Universal Robots PolyScope program: cottonbot.urp

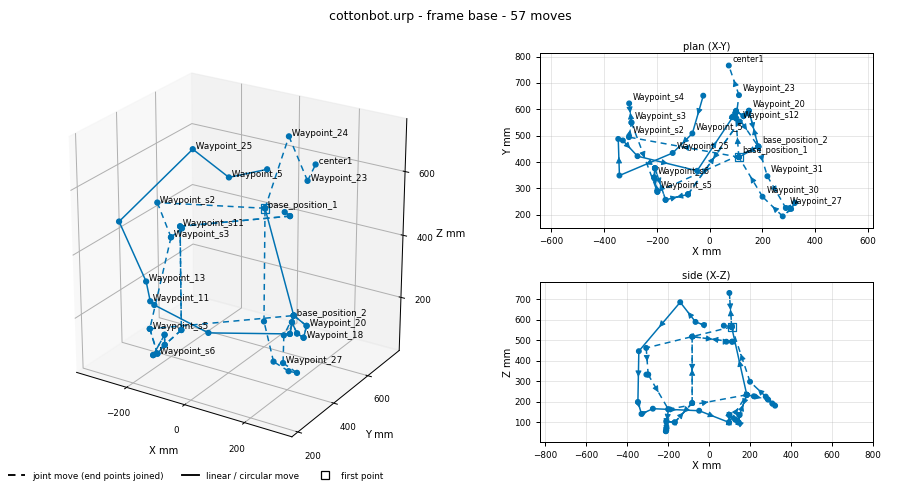
[picture p0: tool path of cottonbot.urp in frame base, 57 of 63 moves have a stored position in this frame; points joined in program order, loops and branches not executed]
Program cottonbot (installation=default directory=/programs/Nicolas_Arteaga/new folder createdIn=5.8.2.10297 lastSavedIn=5.12.4.1101661 robotSerialNumber=20225502378)
Calibrated DH parameters: a=[0.00022, -0.425328, -0.389701, 0.000059, 0.000065, 0]; d=[0.162608, 0.803456, 9.992211, -10.662202, 0.099702, 0.099559]; alpha=[1.570756, 0.001543, 0.004316, 1.570651, -1.570122, 0]; deltaTheta=[0, 0.002917, 0.116094, -0.119008, 0, -0.000001]
Robot Program (runOnlyOnce=true)
  'The whole program merged'
  Timer (action=Start) variable(name=timer_2)
  Timer (action=Start) variable(name=timer_3)
  'Now starts the Sugar Workflow'
  MoveJ speed 60 deg/s, acceleration 80 deg/s^2 (useActiveTCP=true) feature=Base
    Waypoint base_position_1: TCP in base x=110.873 y=418.875 z=565.206 mm, rx=-1.5602 ry=-0.9891 rz=-1.3624 rad; joints [200.91, -129.117, 99.415, 36.172, 41.428, 90] deg; TCP offset x=0 y=0 z=191.5 mm, rx=0 ry=0 rz=0 rad
    Waypoint Waypoint_s2: TCP in base x=-305.749 y=494.617 z=462.545 mm, rx=-1.1337 ry=-1.2693 rz=-1.1298 rad; joints [300.263, -100.211, 102.502, -1.736, 114.115, 89.999] deg; TCP offset x=0 y=0 z=191.5 mm, rx=0 ry=0 rz=0 rad
    URCap Gripper Activate (Robotiq_Grippers, Robotiq Inc.) dataModel(ResetAndActivateKey=false)
    URCap Gripper (Robotiq_Grippers, Robotiq Inc.) dataModel(position=20.0, force=0.0, speed=0.0, positionInDouble=20.0, forceInDouble=0.0, speedInDouble=0.0, slaveIds=[9], blocking=true)
    Waypoint Waypoint_s3: TCP in base x=-296.164 y=549.885 z=332.617 mm, rx=-1.2863 ry=-1.1731 rz=-1.2824 rad; joints [302.576, -85.481, 108.119, -21.976, 128.323, 90.062] deg
    Waypoint Waypoint_s4: TCP in base x=-304.886 y=622.528 z=332.693 mm, rx=-1.2845 ry=-1.1692 rz=-1.2825 rad; joints [298.729, -77.999, 99.501, -20.953, 124.442, 90.195] deg
    URCap Gripper (Robotiq_Grippers, Robotiq Inc.) dataModel(position=35.0, force=100.0, speed=100.0, positionInDouble=35.0, forceInDouble=100.0, speedInDouble=100.0, slaveIds=[9], blocking=true)
    Wait Sleep waitTime=0.5
    URCap Gripper (Robotiq_Grippers, Robotiq Inc.) dataModel(position=0.0, force=100.0, speed=0.0, positionInDouble=0.0, forceInDouble=100.0, speedInDouble=0.0, slaveIds=[9], blocking=true)
    Waypoint Waypoint_s3: TCP in base x=-296.164 y=549.885 z=332.617 mm, rx=-1.2863 ry=-1.1731 rz=-1.2824 rad; joints [302.576, -85.481, 108.119, -21.976, 128.323, 90.062] deg
    Waypoint Waypoint_s5: TCP in base x=-197.91 y=287.3 z=163.432 mm, rx=-1.5535 ry=0.1524 rz=-0.1096 rad; joints [326.967, -91.614, 148.2, -58.357, 156.715, 180] deg; TCP offset x=0 y=0 z=191.5 mm, rx=0 ry=0 rz=0 rad
    URCap Gripper (Robotiq_Grippers, Robotiq Inc.) dataModel(position=50.0, force=100.0, speed=0.0, positionInDouble=50.0, forceInDouble=100.0, speedInDouble=0.0, slaveIds=[9], blocking=true)
    Waypoint Waypoint_s6: TCP in base x=-209.858 y=341.762 z=56.515 mm, rx=-1.5807 ry=0.0548 rz=-0.0662 rad; joints [313.143, -65.937, 152.318, -85.713, 137.744, 180] deg; TCP offset x=0 y=0 z=191.5 mm, rx=0 ry=0 rz=0 rad
    Waypoint Waypoint_s7: TCP in base x=-207.363 y=377.054 z=70.962 mm, rx=-1.5764 ry=0.0343 rz=-0.0374 rad; joints [304.137, -69.797, 152.569, -82.518, 126.942, 179.974] deg; TCP offset x=0 y=0 z=191.5 mm, rx=0 ry=0 rz=0 rad
    URCap Gripper (Robotiq_Grippers, Robotiq Inc.) dataModel(position=100.0, force=100.0, speed=0.0, positionInDouble=100.0, forceInDouble=100.0, speedInDouble=0.0, slaveIds=[9], blocking=true)
    Waypoint Waypoint_s8: TCP in base x=-207.108 y=376.646 z=104.52 mm, rx=-1.5811 ry=0.0321 rz=-0.0396 rad; joints [304.156, -79.665, 151.838, -71.558, 126.955, 180.055] deg
    Waypoint Waypoint_s9: TCP in base x=-166.798 y=256.956 z=99.586 mm, rx=-1.5812 ry=0.0311 rz=-0.0496 rad; joints [323.963, -84.01, 161.527, -76.66, 147.1, 180] deg; TCP offset x=0 y=0 z=191.5 mm, rx=0 ry=0 rz=0 rad
    Waypoint Waypoint_s10: TCP in base x=-81.738 y=277.755 z=193.913 mm, rx=-1.6539 ry=-0.0026 rz=-1.0019 rad; joints [319.07, -96.736, 145.387, -56.678, 176.026, 135] deg; TCP offset x=0 y=0 z=191.5 mm, rx=0 ry=0 rz=0 rad
    Waypoint Waypoint_s11: TCP in base x=-81.724 y=277.748 z=517.554 mm, rx=-1.6566 ry=-0.0181 rz=-1.0161 rad; joints [319.137, -114.467, 104.986, 2.526, 175.909, 135] deg; TCP offset x=0 y=0 z=191.5 mm, rx=0 ry=0 rz=0 rad
    Waypoint Waypoint_s12: TCP in base x=113.097 y=553.265 z=492.993 mm, rx=-1.5561 ry=-0.4924 rz=-0.7353 rad; joints [227.113, -110.707, 105.414, 5.953, 56.661, 135.029] deg; TCP offset x=0 y=0 z=191.5 mm, rx=0 ry=0 rz=0 rad
    Waypoint Waypoint_s13: TCP in base x=85.146 y=570.31 z=492.98 mm, rx=-0.6297 ry=-2.0123 rz=-2.0637 rad; joints [234.679, -108.87, 104.254, 5.245, 64.223, 25.001] deg; TCP offset x=0 y=0 z=191.5 mm, rx=0 ry=0 rz=0 rad
    Waypoint Waypoint_s12: TCP in base x=113.097 y=553.265 z=492.993 mm, rx=-1.5561 ry=-0.4924 rz=-0.7353 rad; joints [227.113, -110.707, 105.414, 5.953, 56.661, 135.029] deg; TCP offset x=0 y=0 z=191.5 mm, rx=0 ry=0 rz=0 rad
    Waypoint Waypoint_s11: TCP in base x=-81.724 y=277.748 z=517.554 mm, rx=-1.6566 ry=-0.0181 rz=-1.0161 rad; joints [319.137, -114.467, 104.986, 2.526, 175.909, 135] deg; TCP offset x=0 y=0 z=191.5 mm, rx=0 ry=0 rz=0 rad
    Waypoint Waypoint_s10: TCP in base x=-81.738 y=277.755 z=193.913 mm, rx=-1.6539 ry=-0.0026 rz=-1.0019 rad; joints [319.07, -96.736, 145.387, -56.678, 176.026, 135] deg; TCP offset x=0 y=0 z=191.5 mm, rx=0 ry=0 rz=0 rad
    Waypoint Waypoint_s9: TCP in base x=-166.798 y=256.956 z=99.586 mm, rx=-1.5812 ry=0.0311 rz=-0.0496 rad; joints [323.963, -84.01, 161.527, -76.66, 147.1, 180] deg; TCP offset x=0 y=0 z=191.5 mm, rx=0 ry=0 rz=0 rad
    Waypoint Waypoint_s8: TCP in base x=-207.108 y=376.646 z=104.52 mm, rx=-1.5811 ry=0.0321 rz=-0.0396 rad; joints [304.156, -79.665, 151.838, -71.558, 126.955, 180.055] deg; TCP offset x=0 y=0 z=191.5 mm, rx=0 ry=0 rz=0 rad
    Waypoint Waypoint_s7: TCP in base x=-207.363 y=377.054 z=70.962 mm, rx=-1.5764 ry=0.0343 rz=-0.0374 rad; joints [304.137, -69.797, 152.569, -82.518, 126.942, 179.974] deg
    URCap Gripper (Robotiq_Grippers, Robotiq Inc.) dataModel(position=0.0, force=0.0, speed=100.0, positionInDouble=0.0, forceInDouble=0.0, speedInDouble=100.0, slaveIds=[9], blocking=true)
    Waypoint Waypoint_s6: TCP in base x=-209.858 y=341.762 z=56.515 mm, rx=-1.5807 ry=0.0548 rz=-0.0662 rad; joints [313.143, -65.937, 152.318, -85.713, 137.744, 180] deg; TCP offset x=0 y=0 z=191.5 mm, rx=0 ry=0 rz=0 rad
    Waypoint Waypoint_s5: TCP in base x=-197.91 y=287.3 z=163.432 mm, rx=-1.5535 ry=0.1524 rz=-0.1096 rad; joints [326.967, -91.614, 148.2, -58.357, 156.715, 180] deg; TCP offset x=0 y=0 z=191.5 mm, rx=0 ry=0 rz=0 rad
    Waypoint base_position_2: TCP in base x=184.715 y=458.614 z=234.006 mm, rx=-1.6866 ry=-0.757 rz=-1.7388 rad; joints [237.954, -104.402, 143.977, -41.546, 99.477, 90] deg; TCP offset x=0 y=0 z=191.5 mm, rx=0 ry=0 rz=0 rad
  'Now starts turning on the machine'
  MoveJ speed 60 deg/s, acceleration 80 deg/s^2 (useActiveTCP=true) feature=Base
    URCap Gripper (Robotiq_Grippers, Robotiq Inc.) dataModel(position=100.0, force=0.0, speed=100.0, positionInDouble=100.0, forceInDouble=0.0, speedInDouble=100.0, slaveIds=[9], blocking=true)
    Waypoint base_position_2: TCP in base x=184.715 y=458.614 z=234.006 mm, rx=-1.6866 ry=-0.757 rz=-1.7388 rad; joints [237.954, -104.402, 143.977, -41.546, 99.477, 90] deg
    Waypoint Waypoint_20: TCP in base x=148.965 y=594.736 z=135.542 mm, rx=-1.534 ry=-0.9908 rz=-1.4978 rad; joints [241.135, -76.483, 134.799, -57.047, 85.473, 90.096] deg; TCP offset x=0 y=0 z=191.5 mm, rx=0 ry=0 rz=0 rad
    Waypoint Waypoint_18: TCP in base x=144.729 y=585.254 z=99.641 mm, rx=-1.6452 ry=-1.0629 rz=-1.3952 rad; joints [240.345, -76.212, 134.041, -48.93, 84.034, 89.956] deg
    Waypoint Waypoint_6: TCP in base x=128.361 y=574.771 z=113.603 mm, rx=-1.6021 ry=-1.0547 rz=-1.4085 rad; joints [240.991, -78.96, 136.832, -51.045, 83.741, 89.995] deg
    Waypoint Waypoint_17: TCP in base x=99.779 y=593.316 z=135.031 mm, rx=-1.492 ry=-1.1083 rz=-1.3373 rad; joints [241.005, -80.644, 135.434, -49.386, 76.736, 90.11] deg
    Waypoint Waypoint_16: TCP in base x=97.63 y=585.581 z=99.564 mm, rx=-1.5888 ry=-1.15 rz=-1.2562 rad; joints [240.815, -78.841, 134.769, -44.332, 76.722, 90.097] deg
    Waypoint base_position_2: TCP in base x=184.715 y=458.614 z=234.006 mm, rx=-1.6866 ry=-0.757 rz=-1.7388 rad; joints [237.954, -104.402, 143.977, -41.546, 99.477, 90] deg; TCP offset x=0 y=0 z=191.5 mm, rx=0 ry=0 rz=0 rad
  'Now the stick Placement'
  MoveJ speed 60 deg/s, acceleration 80 deg/s^2 (useActiveTCP=true) feature=Base
    Waypoint base_position_2: TCP in base x=184.715 y=458.614 z=234.006 mm, rx=-1.6866 ry=-0.757 rz=-1.7388 rad; joints [237.954, -104.402, 143.977, -41.546, 99.477, 90] deg
    URCap Gripper Activate (Robotiq_Grippers, Robotiq Inc.) dataModel(ResetAndActivateKey=false)
    URCap Gripper (Robotiq_Grippers, Robotiq Inc.) dataModel(position=70.0, force=0.0, speed=100.0, positionInDouble=70.0, forceInDouble=0.0, speedInDouble=100.0, slaveIds=[9], blocking=true)
    Waypoint Waypoint_31: TCP in base x=219.073 y=346.37 z=226.939 mm, rx=-1.0793 ry=1.1503 rz=-0.4496 rad; joints [242.985, -108.839, 146.791, -38.8, 126.314, 210] deg; TCP offset x=0 y=0 z=191.5 mm, rx=0 ry=0 rz=0 rad
    Waypoint Waypoint_27: TCP in base x=288.911 y=225.994 z=210.348 mm, rx=-0.5682 ry=1.4712 rz=-0.493 rad; joints [230.777, -108.395, 149.908, -42.839, 137.738, 230] deg; TCP offset x=0 y=0 z=191.5 mm, rx=0 ry=0 rz=0 rad
    Waypoint stick1: TCP in base x=322.798 y=244.707 z=180.935 mm, rx=-0.6006 ry=1.5021 rz=-0.5325 rad; joints [227.883, -97.858, 147.006, -47.332, 135.838, 229.943] deg; TCP offset x=0 y=0 z=191.5 mm, rx=0 ry=0 rz=0 rad
    URCap Gripper (Robotiq_Grippers, Robotiq Inc.) dataModel(position=100.0, force=0.0, speed=0.0, positionInDouble=100.0, forceInDouble=0.0, speedInDouble=0.0, slaveIds=[9], blocking=true)
    Waypoint Waypoint_3: TCP in base x=308.934 y=222.719 z=191.895 mm, rx=-0.6005 ry=1.5021 rz=-0.5324 rad; joints [226.032, -105.235, 149.7, -42.849, 134.017, 229.721] deg
    Waypoint Waypoint_4: TCP in base x=277.219 y=194.361 z=225.221 mm, rx=-0.5767 ry=1.5048 rz=-0.5799 rad; joints [231.096, -114.882, 148.99, -33.185, 141.571, 228.474] deg
    Waypoint Waypoint_30: TCP in base x=200.562 y=268.796 z=297.612 mm, rx=-1.3009 ry=0.8471 rz=-0.8634 rad; joints [232.325, -138.788, 148.891, -15.287, 116.251, 180] deg; TCP offset x=0 y=0 z=191.5 mm, rx=0 ry=0 rz=0 rad
    Waypoint Waypoint_28: TCP in base x=110.872 y=418.885 z=565.169 mm, rx=-1.6121 ry=0.3611 rz=-0.2078 rad; joints [200.913, -129.115, 99.418, 36.172, 41.428, 180] deg; TCP offset x=0 y=0 z=191.5 mm, rx=0 ry=0 rz=0 rad
    Waypoint Waypoint_24: TCP in base x=99.712 y=565.5 z=730.734 mm, rx=-1.4619 ry=0.2517 rz=-0.2966 rad; joints [243.031, -99.822, 65.521, 28.761, 83.192, 180] deg; TCP offset x=0 y=0 z=191.5 mm, rx=0 ry=0 rz=0 rad
    Waypoint Waypoint_23: TCP in base x=111.331 y=653.695 z=566.749 mm, rx=-1.7943 ry=0.2693 rz=-0.1351 rad; joints [243.037, -87.632, 65.808, 35.91, 77.265, 180] deg; TCP offset x=0 y=0 z=191.5 mm, rx=0 ry=0 rz=0 rad
    Waypoint center1: TCP in base x=72.723 y=766.045 z=571.175 mm, rx=-1.5688 ry=-0.0203 rz=0.0146 rad; joints [244.553, -79.065, 65.7, 13.074, 63.165, 180.144] deg; TCP offset x=0 y=0 z=191.5 mm, rx=0 ry=0 rz=0 rad
  'Now Cotton Candy Creation'
  SuppressedNode
    radius := 0.149
  radius := 0.13
  height := 0.05
  SuppressedNode
    cold_start_wait := 101.25
  SuppressedNode
    start_wait := GP_int_in[0]
  SuppressedNode
    start_time := GP_int_in[1]
  SuppressedNode
    circle_time := GP_int_in[2]
  start_wait := 1
  start_time := 33.75
  circle_time := 3.75
  SuppressedNode
    cold_start_spin := 28
  SuppressedNode
    cold_start_spin := 100
  center := Joint_6_name
  bottom := pose_add(center, p[0, -radius, height, 0, 0, 0])
  right := pose_add(center, p[-radius, 0, -height, 0, 0, 0])
  top_circ := pose_add(center, p[0, radius, height, 0, 0, 0])
  left := pose_add(center, p[radius, 0, -height, 0, 0, 0])
  SuppressedNode
    diff := pose_sub(left,bottom )
  SuppressedNode
    Loop While (checkContinuously=false) expression=circles_no>0
      MoveP speed 250 mm/s, acceleration 1200 mm/s^2 (blendRadius=0.125 useActiveTCP=true) feature=Base
        Waypoint Waypoint (Variable): variable(name=bottom)
        CircleMove (OrientationMode=UNCONSTRAINED)
          Waypoint Waypoint (Variable): variable=left
          Waypoint Waypoint (Variable): variable(name=top_circ)
      MoveP speed 250 mm/s, acceleration 1200 mm/s^2 (blendRadius=0.025 useActiveTCP=true) feature=Base
        Waypoint Waypoint (Variable): variable=top_circ
        CircleMove (OrientationMode=UNCONSTRAINED)
          Waypoint Waypoint (Variable): variable=right
          Waypoint Waypoint (Variable): variable=bottom
      circles_no := circles_no-1
  Timer (action=Stop) variable=timer_3
  SuppressedNode
    Wait Sleep waitTime=101.25
  SuppressedNode
    Wait Condition expression=GP_int_in[0]
  Script: sleep(start_wait)
  Timer (action=Start) variable(name=timer_1)
  Loop While (checkContinuously=false) expression=start_time>0
    MoveP speed 250 mm/s, acceleration 1200 mm/s^2 (blendRadius=0.125 useActiveTCP=true) feature=Base
      Waypoint Waypoint (Variable): variable=bottom
      CircleMove (OrientationMode=UNCONSTRAINED)
        Waypoint Waypoint (Variable): variable=left
        Waypoint Waypoint (Variable): variable=top_circ
    MoveP speed 250 mm/s, acceleration 1200 mm/s^2 (blendRadius=0.025 useActiveTCP=true) feature=Base
      Waypoint Waypoint (Variable): variable=top_circ
      CircleMove (OrientationMode=UNCONSTRAINED)
        Waypoint Waypoint (Variable): variable=right
        Waypoint Waypoint (Variable): variable=bottom
    SuppressedNode
      bottom := pose_add(bottom, p[0, 0, height/(cold_start_spin/2), 0, 0, 0])
    SuppressedNode
      right := pose_add(left, p[0, 0, 2*height/cold_start_spin, 0, 0, 0])
    SuppressedNode
      top_circ := pose_add(top_circ, p[0, 0, 2*height/cold_start_spin, 0, 0, 0])
    SuppressedNode
      left := pose_add(left, p[0, 0, 2*height/cold_start_spin, 0, 0, 0])
    start_time := start_time-circle_time
  Timer (action=Stop) variable=timer_1
  MoveL speed 250 mm/s, acceleration 1200 mm/s^2 (useActiveTCP=true) feature=Base
    Waypoint Waypoint_2: TCP in base x=-24.03 y=651.793 z=574.352 mm, rx=-0.9882 ry=-1.0644 rz=-1.2372 rad; joints [248.909, -99.854, 96.502, -11.42, 64.977, 96.89] deg
    Waypoint Waypoint_5: TCP in base x=-65.345 y=508.583 z=589.478 mm, rx=-0.8529 ry=-1.3704 rz=-1.3892 rad; joints [239.18, -119.542, 101.662, 8.745, 51.039, 78.082] deg
    Waypoint Waypoint_25: TCP in base x=-139.92 y=434.562 z=685.517 mm, rx=0.2728 ry=-1.6358 rz=-2.1043 rad; joints [228.521, -129.991, 99.843, -7.046, 27.223, 41.249] deg
    Waypoint Waypoint_12: TCP in base x=-341.731 y=349.139 z=446.744 mm, rx=1.0197 ry=-1.4327 rz=-1.9509 rad; joints [261.046, -128.059, 128.66, -21.395, 27.658, 2.719] deg
    Waypoint Waypoint_13: TCP in base x=-346.288 y=487.83 z=199.367 mm, rx=1.1258 ry=-1.8238 rz=-1.9724 rad; joints [274.508, -89.471, 132.703, -38.479, 53.378, -24.773] deg
    Waypoint Waypoint_11: TCP in base x=-328.73 y=482.036 z=140.622 mm, rx=1.1107 ry=-1.8448 rz=-1.9801 rad; joints [271.637, -83.004, 138.617, -50.548, 51.741, -25.068] deg
    URCap Gripper Activate (Robotiq_Grippers, Robotiq Inc.) dataModel(ResetAndActivateKey=false)
    URCap Gripper (Robotiq_Grippers, Robotiq Inc.) dataModel(position=0.0, force=0.0, speed=100.0, positionInDouble=0.0, forceInDouble=0.0, speedInDouble=100.0, slaveIds=[9], blocking=true)
    Waypoint Waypoint_14: TCP in base x=-273.276 y=422.463 z=166.295 mm, rx=0.9524 ry=-2.167 rz=-1.9141 rad; joints [271.624, -104.005, 143.852, -26.72, 64.174, -25.036] deg
    URCap Gripper (Robotiq_Grippers, Robotiq Inc.) dataModel(position=100.0, force=0.0, speed=100.0, positionInDouble=100.0, forceInDouble=0.0, speedInDouble=100.0, slaveIds=[9], blocking=true)
    MoveL speed 250 mm/s, acceleration 1200 mm/s^2 (useActiveTCP=true) feature=Base
      Waypoint Waypoint_15: TCP in base x=-47.378 y=367.135 z=156.328 mm, rx=-1.8568 ry=-1.4579 rz=-0.9844 rad; joints [256.209, -119.497, 138.801, 14.851, 90.035, 90] deg; TCP offset x=0 y=0 z=191.5 mm, rx=0 ry=0 rz=0 rad
      Waypoint Waypoint_16: TCP in base x=97.63 y=585.581 z=99.564 mm, rx=-1.5888 ry=-1.15 rz=-1.2562 rad; joints [240.815, -78.841, 134.769, -44.332, 76.722, 90.097] deg; TCP offset x=0 y=0 z=191.5 mm, rx=0 ry=0 rz=0 rad
      Waypoint Waypoint_17: TCP in base x=99.779 y=593.316 z=135.031 mm, rx=-1.492 ry=-1.1083 rz=-1.3373 rad; joints [241.005, -80.644, 135.434, -49.386, 76.736, 90.11] deg
      Waypoint Waypoint_6: TCP in base x=128.361 y=574.771 z=113.603 mm, rx=-1.6021 ry=-1.0547 rz=-1.4085 rad; joints [240.991, -78.96, 136.832, -51.045, 83.741, 89.995] deg
      Waypoint Waypoint_18: TCP in base x=144.729 y=585.254 z=99.641 mm, rx=-1.6452 ry=-1.0629 rz=-1.3952 rad; joints [240.345, -76.212, 134.041, -48.93, 84.034, 89.956] deg
      Timer (action=Stop) variable=timer_2
      SuppressedNode
        Wait Sleep waitTime=90
      Script: sleep(5)
      Waypoint Waypoint_20: TCP in base x=148.965 y=594.736 z=135.542 mm, rx=-1.534 ry=-0.9908 rz=-1.4978 rad; joints [241.135, -76.483, 134.799, -57.047, 85.473, 90.096] deg
      Waypoint base_position_2: TCP in base x=184.715 y=458.614 z=234.006 mm, rx=-1.6866 ry=-0.757 rz=-1.7388 rad; joints [237.954, -104.402, 143.977, -41.546, 99.477, 90] deg; TCP offset x=0 y=0 z=191.5 mm, rx=0 ry=0 rz=0 rad
      Waypoint Waypoint_22: TCP in base x=110.871 y=418.877 z=565.218 mm, rx=-1.5321 ry=-1.0694 rz=-1.423 rad; joints [200.91, -129.118, 99.415, 36.169, 41.427, 84.919] deg; TCP offset x=0 y=0 z=191.5 mm, rx=0 ry=0 rz=0 rad
      Waypoint base_position_1: TCP in base x=110.873 y=418.875 z=565.206 mm, rx=-1.5602 ry=-0.9891 rz=-1.3624 rad; joints [200.91, -129.117, 99.415, 36.172, 41.428, 90] deg; TCP offset x=0 y=0 z=191.5 mm, rx=0 ry=0 rz=0 rad
